ABB RobotStudio station: RobMan2.rsstn

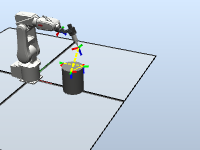
Station RobMan1 (saved by RobotStudio 6.6.7701.1025)
Controller Sistema1
  mechanical unit ROB_1: IRB120_3_58__01, 6 joints, base frame (0, 0, 0) mm
Layout (positions relative to the parent item):
  - IRB120_3_58__01 [mechanism, from Robots\IRB120_3_58_G_01.rslib] at (0, 0, 0) mm; joint values [0, 0, 0, 0, 0.5236, 0] (rad or m)
  - MyTool [mechanism, from Training Objects\myTool.rslib] at (364.35, 0, 594) mm, rotated rx 180 ry 60 rz 180 deg
  - Pieza_1 [part]
Attachment: MyTool is attached to IRB120_3_58__01 / Link6
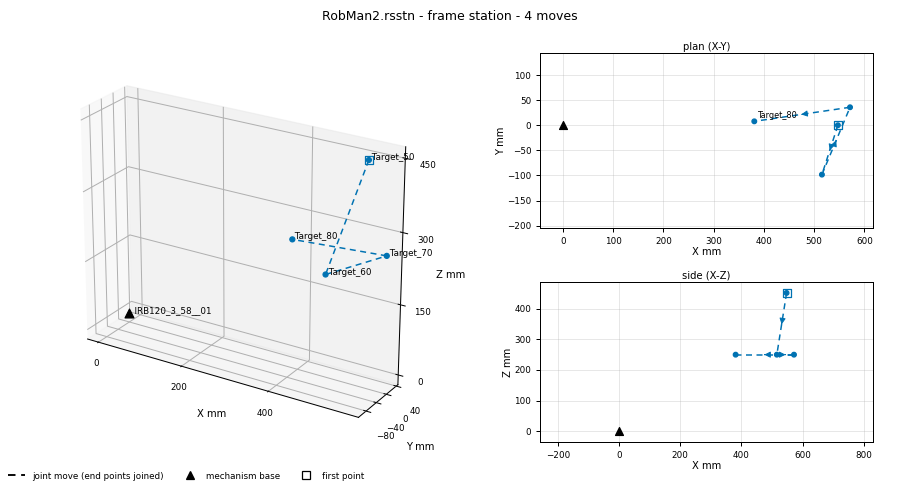
[picture p0: tool path of RobMan2.rsstn in frame station, 4 of 4 moves have a stored position in this frame; points joined in program order, loops and branches not executed]
Targets, tools, work objects and paths stored in the station, written as RAPID:
! task T_ROB1
MODULE CalibData
  PERS tooldata MyTool:=[TRUE,[[31.792631019,0,229.638935148],[0.945518576,0,0.325568154,0]],[1,[0,0,1],[1,0,0,0],0,0,0]];
ENDMODULE

! task T_ROB1
MODULE Module1
  CONST robtarget Target_50:=[[547.330665099,0,451.64730631],[0.190808996,0,0.981627183,0],[-1,0,-1,0],[9E+09,9E+09,9E+09,9E+09,9E+09,9E+09]];
  CONST robtarget Target_60:=[[515.556908903,-98.297458162,250],[0,0.983647442,0.180104717,0],[0,0,0,0],[9E+09,9E+09,9E+09,9E+09,9E+09,9E+09]];
  CONST robtarget Target_70:=[[571.527992386,35.779676541,250],[0,0.545139081,0.838345622,0],[0,0,0,0],[9E+09,9E+09,9E+09,9E+09,9E+09,9E+09]];
  CONST robtarget Target_80:=[[380.916310122,7.770311733,250],[0,-0.661228736,0.75018435,0],[0,0,0,0],[9E+09,9E+09,9E+09,9E+09,9E+09,9E+09]];
  PROC Path_10()
    MoveJ Target_50,v1000,fine,MyTool\WObj:=wobj0;
    MoveJ Target_60,v1000,fine,MyTool\WObj:=wobj0;
    MoveJ Target_70,v1000,fine,MyTool\WObj:=wobj0;
    MoveJ Target_80,v1000,fine,MyTool\WObj:=wobj0;
  ENDPROC
ENDMODULE

